{attribute 'GeneratedUsingTerminal: EK1122-0000-0018'}
{attribute addProperty BoxType "EK1122-0000-0018"}
{attribute addProperty Id "Beckhoff_EL72xxsub_EK1100EK1100_1FC0878B2"}
{attribute addProperty CRC "2800219486"}
{attribute addProperty Size "2"}
TYPE Beckhoff_EL72xxEK1122_A6E7F55E EXTENDS EK1122_1FC0878B :
STRUCT
	{attribute addProperty Name "Beckhoff_EL72xxsub_EK1100"}
	{attribute addProperty PreviousPort "Beckhoff EL72xxEK1122 : D"}
	Beckhoff_EL72xxsub_EK1100 : EK1100_1FC0878B;
END_STRUCT
END_TYPE

(* stored: Version 1.2.0.0, ProductVersion 3.1.4024.9
   DUT Beckhoff_EL72xxEK1122_A6E7F55E: Id {718c8ec1-0426-4803-90fc-97e6ea4d88d6} *)
